FUNCTION F_Select : INT
VAR_INPUT
	i_In1			:BOOL;
	i_In2			:BOOL;
	i_In3			:BOOL;
	i_In4			:BOOL;
	i_In5			:BOOL;
END_VAR
VAR
END_VAR

IF i_In1 THEN
	F_Select:=0;
END_IF
IF i_In2 THEN
	F_Select:=1;
END_IF
IF i_In3 THEN
	F_Select:=2;
END_IF
IF i_In4 THEN
	F_Select:=3;
END_IF
IF i_In5 THEN
	F_Select:=4;
END_IF

END_FUNCTION

(* stored: Version 1.1.0.1, ProductVersion 3.1.4024.12
   POU F_Select: Id {319899ee-9f06-467f-a11b-f818e22a2c3b}, SpecialFunc None *)
